FUNCTION_BLOCK FB_INTEGRATE (* Basic Function Block Type *)
  (* Standard: 61499-2 *)
  (* Version 0.0, 2011-07-12, 4DIAC-IDE, 4DIAC-Consortium *)
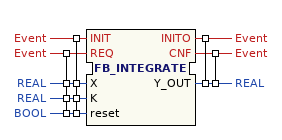
  EVENT_INPUT
    INIT WITH X, K, reset; (* Initialization Request *)
    REQ WITH X, K, reset; (* Normal Execution Request *)
  END_EVENT
  EVENT_OUTPUT
    INITO WITH Y_OUT; (* Initialization Confirm *)
    CNF WITH Y_OUT; (* Execution Confirmation *)
  END_EVENT
  VAR_INPUT
    X : REAL; (* Input value on x-axis *)
    K : REAL := 1.0; (* Factor *)
    reset : BOOL; (* If reset is true Y_OUT is 0 *)
  END_VAR
  VAR_OUTPUT
    Y_OUT : REAL; (* Output value on y-axis *)
  END_VAR
  VAR
    X_last : REAL; (* The last value on x-axis *)
    last : DWORD; (* The last time *)
    tx : DWORD; (* The time in milliseconds *)
    Y_intern : REAL; (* The value on y-axis *)
  END_VAR
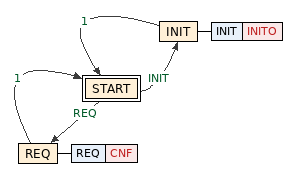
  EC_STATES
    START; (* Initial State *)
    INIT : INIT -> INITO; (* Initialization *)
    REQ : REQ -> CNF; (* Normal execution *)
  END_STATES
  EC_TRANSITIONS
    START TO INIT := INIT;
    INIT TO START := 1;
    START TO REQ := REQ;
    REQ TO START := 1;
  END_TRANSITIONS
  ALGORITHM INIT IN ST: (* Initialization algorithm *)
X_last := X;
  END_ALGORITHM
  ALGORITHM REQ IN ST: (* Normally executed algorithm *)
IF reset THEN
	Y_intern := 0.0;
ELSE
	tx := T_PLC_MS();
	Y_intern := (X + X_last) * 0.5E-3 * DWORD_TO_REAL(tx - last) * K +  Y_intern;
	X_last := X;
	last := tx;
END_IF;

Y_OUT := Y_intern;
  END_ALGORITHM
END_FUNCTION_BLOCK
